FUNCTION_BLOCK PropotionalValve
VAR_INPUT
END_VAR
VAR_OUTPUT
END_VAR
VAR
	//Hardware
	AO_SetPressure AT %Q* : INT;
END_VAR

PROPERTY Pressure : INT
SET
AO_SetPressure := Pressure;
END_SET
END_PROPERTY

END_FUNCTION_BLOCK

(* stored: Version 1.1.0.1, ProductVersion 3.1.4024.9
   POU PropotionalValve: Id {5b85e889-82b8-4c25-8b3a-ea9ac4cc4e30}, SpecialFunc None
   Property Pressure: Id {419427f6-2b16-4457-9e6d-8b72af4c3f15}
   Set Set: Id {894b5635-5846-4a35-b9cc-1ff7b586da00} *)
